// TIA Portal V16 export
// export: Created 2023-08-28T09:37:36.7206819Z, ExportSetting WithDefaults, DisplayName Totally Integrated Automation Portal, DisplayVersion V16 Update 6, DisplayName TIA Portal Version Control Interface, DisplayVersion V16 Update 2, DisplayName TIA Portal Openness, DisplayVersion V16 Update 6, DisplayName STEP 7 Professional, DisplayVersion V16 Update 6, DisplayName STEP 7 Safety, DisplayVersion V16, DisplayName WinCC Advanced, DisplayVersion V16 Update 6
DATA_BLOCK "dbmanagement"   // DB91
TITLE = instacja zarz adzająca
{ S7_Optimized_Access := 'FALSE' }
AUTHOR : rtecmer
VERSION : 0.1
// blok danych pośrednicząc  pomiędzy warstwami
// stored: AutoNumber true, DBAccessibleFromOPCUA true, IsOnlyStoredInLoadMemory false, IsWriteProtectedInAS false
   VAR
      reset : Struct
         resetLicznikPracy_P1 : Bool;   // kasawanie licznika pracy
         resetLicznikPracy_P2 : Bool;   // kasawanie licznika pracy
         resetLicznikPracy_P3 : Bool;   // kasawanie licznika pracy
         resetLicznikPracy_P4 : Bool;   // kasawanie licznika pracy
      END_STRUCT;
      sterowanie_1 : Struct
         stop_falownik : Bool;   // zatrzymanie sterowania falownikiem
         tryb_automat : Bool;   // bit sygnalizacji pracy w automacie zestawu
         "alarm-warning" : Bool;   // alarm ostrzerzenie
         "alarm-modbus" : Bool;   // alarm modbus
         alarm_comunication_WinCC : Bool;   // alarm kominikacji wincc
         "alarm-comunication_HMI" : Bool;
         awaria_modbus_falownik : Bool;   // na potrzeby indentyfikacji awarii do tabeli alarów
         awaria_modbus_przepływ_pomp : Bool;   // na potrzeby indentyfikacji awarii do tabeli alarów
         awaria_modbus_przepływ_magist : Bool;   // na potrzeby indentyfikacji awarii do tabeli alarów
         awaria_modbus_mt101 : Bool;   // na potrzeby indentyfikacji awarii do tabeli alarów
         aktywna_P1 : Bool;
         aktywna_P2 : Bool;
         aktywna_P3 : Bool;
         aktywna_P4 : Bool;
         aktywna_Z11 : Bool;
         aktywna_Z12 : Bool;
         tempStrategia_pompownia : Int;   // Słowo tymczasowe przechwycone podczas wystapienia awarii niskiego ciśnienia magistrala
      END_STRUCT;
      awaria_falownika_F1 : Bool;   // Gotowość falownika 1
      awaria_falownika_F2 : Bool;   // Gotowość falownika 2
      brak_zasilania_RS : Bool;   // Brak zasilania
      instHourStart_Filling : Real;   // Godzina start napełniania
      instHourStop_Filling : Real;   // Godzina stop napełniania
      instHourStart_City : Real;   // Godzina start przetłaczanie miasto DN225
      instHourStop_City : Real;   // Godzina stop przetłaczanie miasto DN225
      instHourStart_Replen : Real;   // Godzina start dosilanie DN500
      instHourStop_Replen : Real;   // Godzina stop dosilanie DN500
      "Alarm analogs to HMI" : Struct   // Alarmy analogowe dla HMI
         "B5 Magistrala max" : Real := 8.5;   // alarm max
         "B6 Miasto max" : Real := 8.0;   // alarm max
         "B7 Pompownia max" : Real := 8.0;   // alarm max
         "B8 suchonieg min" : Real := 0.5;   // alarm min
         "Zbiornik max Nr_1" : Real := 558.0;   // alarm max
         "Zbiornik max Nr_2" : Real := 558.0;   // alarm max
         "Zbiornik max Nr_3" : Real := 558.0;   // alarm max
         "Zbiornik max Nr_4" : Real := 558.0;   // alarm max
      END_STRUCT;
   END_VAR
BEGIN
END_DATA_BLOCK
